% RSLogix 500 project HB_3_Filler.RSS, saved by version 12.00.00.00 %
PROJECT "PLC"    % processor: MicroLogix 1400 %

PROGRAM FILES
  LAD 2   23 rungs
  LAD 9   42 rungs
  LAD 11   37 rungs
  LAD 12   16 rungs
  LAD 14   17 rungs

DATA FILES
  O0 OUTPUT  7 elements
  I1 INPUT  9 elements
  S2 STATUS  66 elements
  B3 BINARY  14 elements
  T4 TIMER  22 elements
  C5 COUNTER  10 elements
  R6 CONTROL  5 elements
  N7 INTEGER  50 elements
  F8 FLOAT  40 elements
  B11   5 elements
  B12   10 elements
  B13   10 elements
  B23   30 elements
  T24   90 elements
  C25   10 elements
  N27   200 elements
  F28   40 elements

LADDER 2
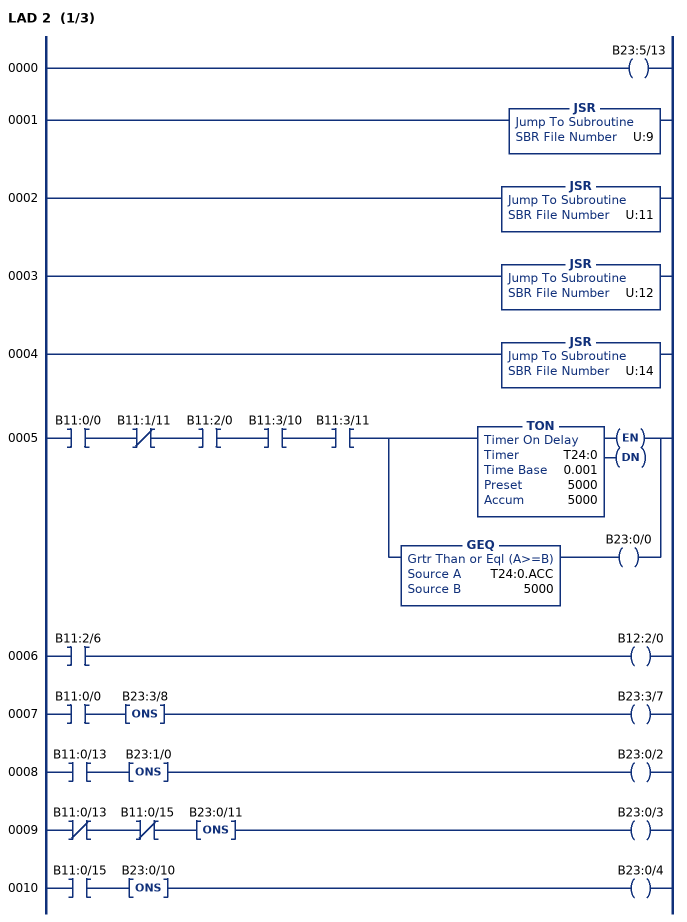
% Rung: 0 %
SOR OTE B23:5/13 EOR
% Rung: 1 %
SOR JSR U:9 EOR
% Rung: 2 %
SOR JSR U:11 EOR
% Rung: 3 %
SOR JSR U:12 EOR
% Rung: 4 %
SOR JSR U:14 EOR
% Rung: 5 %
SOR XIC B11:0/0 XIO B11:1/11 XIC B11:2/0 XIC B11:3/10 XIC B11:3/11 BST TON T24:0 0.001 5000 5000 NXB GEQ T24:0.ACC 5000 OTE B23:0/0 BND EOR
% Rung: 6 %
SOR XIC B11:2/6 OTE B12:2/0 EOR
% Rung: 7 %
SOR XIC B11:0/0 ONS B23:3/8 OTE B23:3/7 EOR
% Rung: 8 %
SOR XIC B11:0/13 ONS B23:1/0 OTE B23:0/2 EOR
% Rung: 9 %
SOR XIO B11:0/13 XIO B11:0/15 ONS B23:0/11 OTE B23:0/3 EOR
% Rung: 10 %
SOR XIC B11:0/15 ONS B23:0/10 OTE B23:0/4 EOR

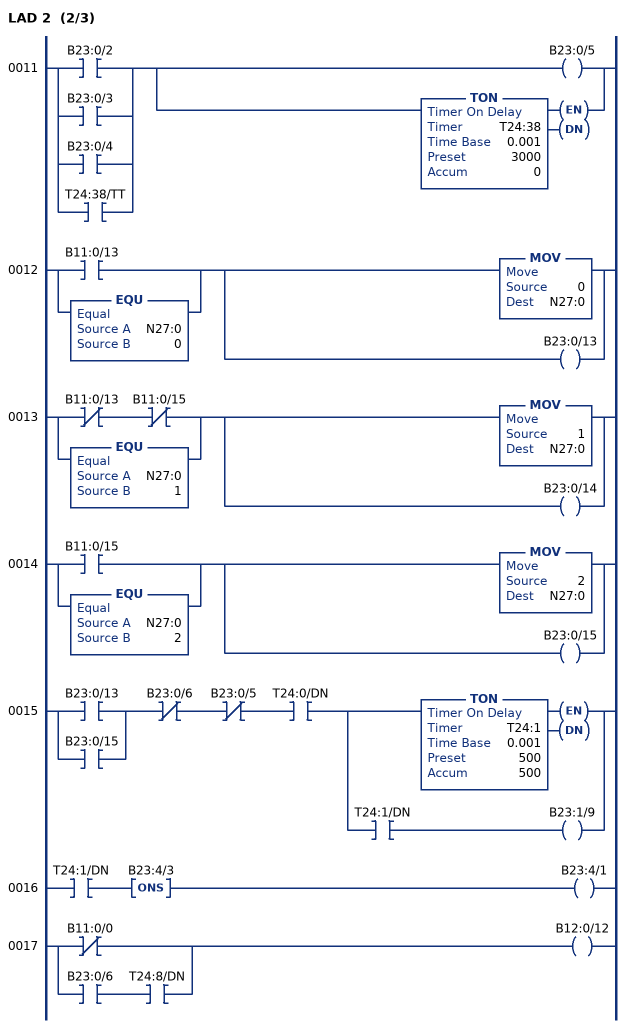
% Rung: 11 %
SOR BST XIC B23:0/2 NXB XIC B23:0/3 NXB XIC B23:0/4 NXB XIC T24:38/TT BND BST OTE B23:0/5 NXB TON T24:38 0.001 3000 0 BND EOR
% Rung: 12 %
SOR BST XIC B11:0/13 NXB EQU N27:0 0 BND BST MOV 0 N27:0 NXB OTE B23:0/13 BND EOR
% Rung: 13 %
SOR BST XIO B11:0/13 XIO B11:0/15 NXB EQU N27:0 1 BND BST MOV 1 N27:0 NXB OTE B23:0/14 BND EOR
% Rung: 14 %
SOR BST XIC B11:0/15 NXB EQU N27:0 2 BND BST MOV 2 N27:0 NXB OTE B23:0/15 BND EOR
% Rung: 15 %
SOR BST XIC B23:0/13 NXB XIC B23:0/15 BND XIO B23:0/6 XIO B23:0/5 XIC T24:0/DN BST TON T24:1 0.001 500 500 NXB XIC T24:1/DN OTE B23:1/9 BND EOR
% Rung: 16 %
SOR XIC T24:1/DN ONS B23:4/3 OTE B23:4/1 EOR
% Rung: 17 %
SOR BST XIO B11:0/0 NXB XIC B23:0/6 XIC T24:8/DN BND OTE B12:0/12 EOR

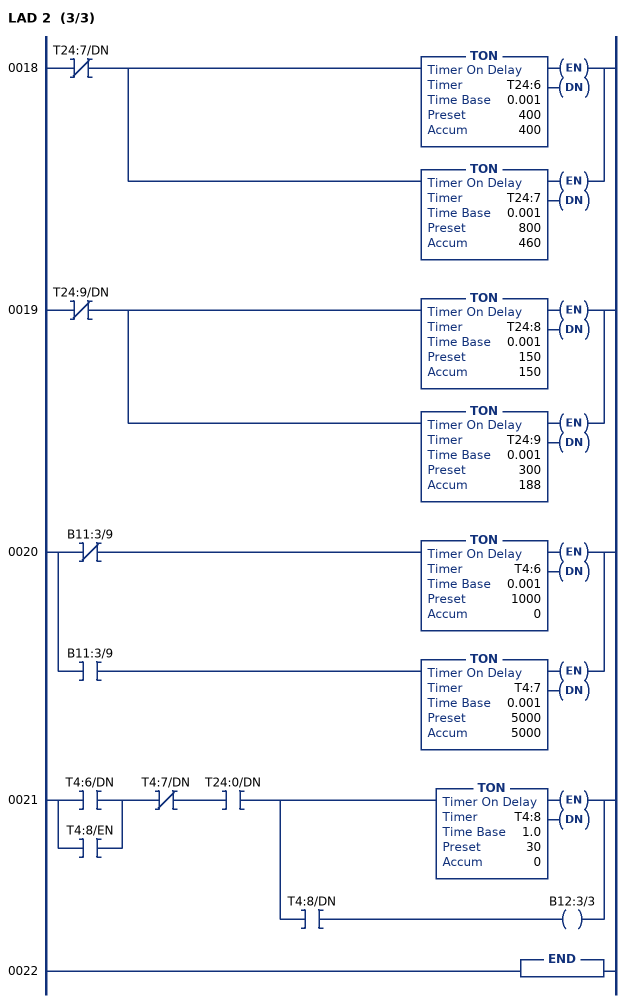
% Rung: 18 %
SOR XIO T24:7/DN BST TON T24:6 0.001 400 400 NXB TON T24:7 0.001 800 460 BND EOR
% Rung: 19 %
SOR XIO T24:9/DN BST TON T24:8 0.001 150 150 NXB TON T24:9 0.001 300 188 BND EOR
% Rung: 20 %
SOR BST XIO B11:3/9 TON T4:6 0.001 1000 0 NXB XIC B11:3/9 TON T4:7 0.001 5000 5000 BND EOR
% Rung: 21 %
SOR BST XIC T4:6/DN NXB XIC T4:8/EN BND XIO T4:7/DN XIC T24:0/DN BST TON T4:8 1.0 30 0 NXB XIC T4:8/DN OTE B12:3/3 BND EOR
% Rung: 22 %
SOR END EOR

LADDER 9
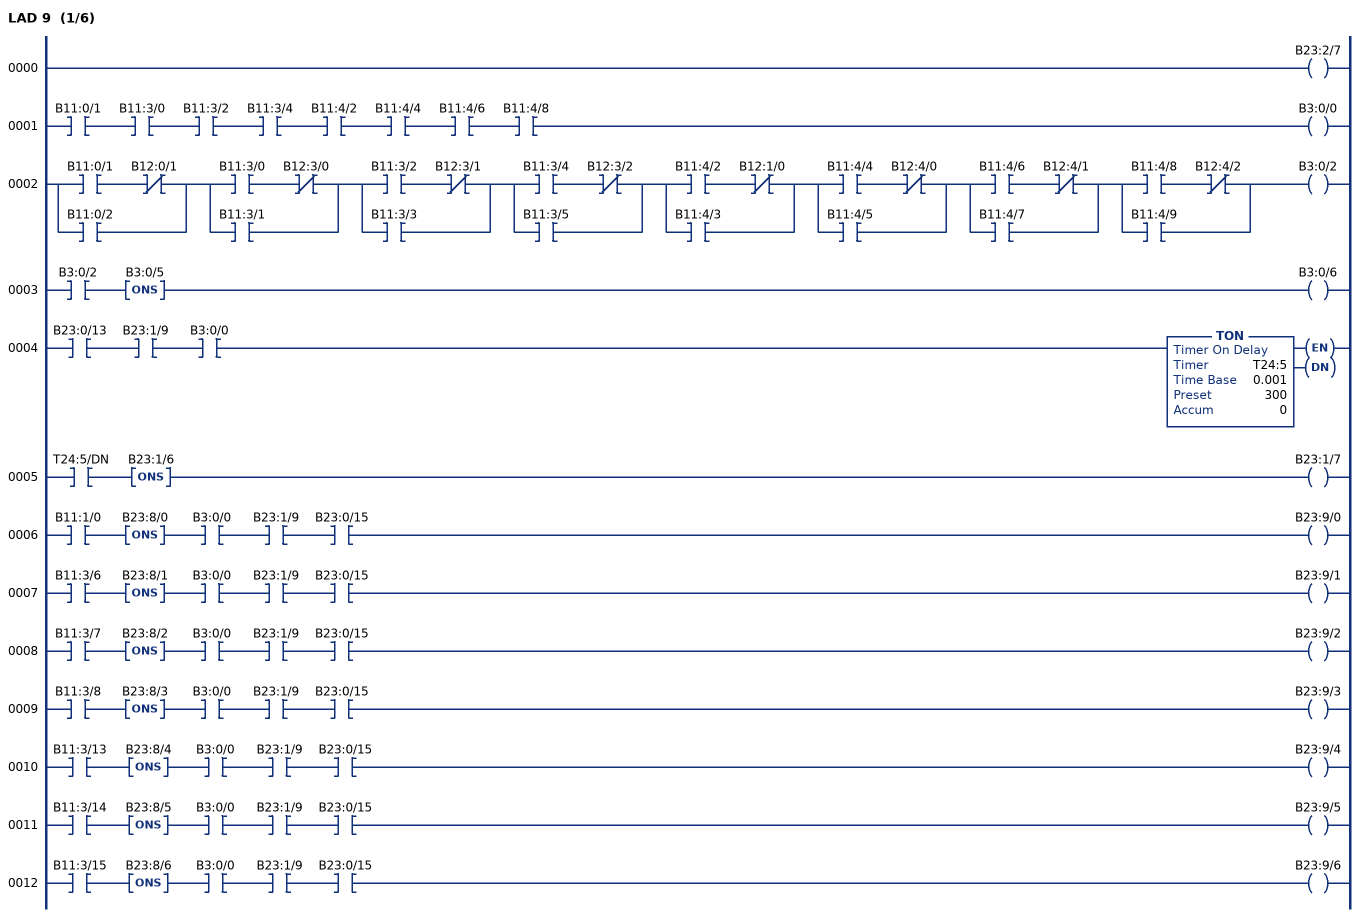
% Rung: 0 %
SOR OTE B23:2/7 EOR
% Rung: 1 %
SOR XIC B11:0/1 XIC B11:3/0 XIC B11:3/2 XIC B11:3/4 XIC B11:4/2 XIC B11:4/4 XIC B11:4/6 XIC B11:4/8 OTE B3:0/0 EOR
% Rung: 2 %
SOR BST XIC B11:0/1 XIO B12:0/1 NXB XIC B11:0/2 BND BST XIC B11:3/0 XIO B12:3/0 NXB XIC B11:3/1 BND BST XIC B11:3/2 XIO B12:3/1 NXB XIC B11:3/3 BND BST XIC B11:3/4 XIO B12:3/2 NXB XIC B11:3/5 BND BST XIC B11:4/2 XIO B12:1/0 NXB XIC B11:4/3 BND BST XIC B11:4/4 XIO B12:4/0 NXB XIC B11:4/5 BND BST XIC B11:4/6 XIO B12:4/1 NXB XIC B11:4/7 BND BST XIC B11:4/8 XIO B12:4/2 NXB XIC B11:4/9 BND OTE B3:0/2 EOR
% Rung: 3 %
SOR XIC B3:0/2 ONS B3:0/5 OTE B3:0/6 EOR
% Rung: 4 %
SOR XIC B23:0/13 XIC B23:1/9 XIC B3:0/0 TON T24:5 0.001 300 0 EOR
% Rung: 5 %
SOR XIC T24:5/DN ONS B23:1/6 OTE B23:1/7 EOR
% Rung: 6 %
SOR XIC B11:1/0 ONS B23:8/0 XIC B3:0/0 XIC B23:1/9 XIC B23:0/15 OTE B23:9/0 EOR
% Rung: 7 %
SOR XIC B11:3/6 ONS B23:8/1 XIC B3:0/0 XIC B23:1/9 XIC B23:0/15 OTE B23:9/1 EOR
% Rung: 8 %
SOR XIC B11:3/7 ONS B23:8/2 XIC B3:0/0 XIC B23:1/9 XIC B23:0/15 OTE B23:9/2 EOR
% Rung: 9 %
SOR XIC B11:3/8 ONS B23:8/3 XIC B3:0/0 XIC B23:1/9 XIC B23:0/15 OTE B23:9/3 EOR
% Rung: 10 %
SOR XIC B11:3/13 ONS B23:8/4 XIC B3:0/0 XIC B23:1/9 XIC B23:0/15 OTE B23:9/4 EOR
% Rung: 11 %
SOR XIC B11:3/14 ONS B23:8/5 XIC B3:0/0 XIC B23:1/9 XIC B23:0/15 OTE B23:9/5 EOR
% Rung: 12 %
SOR XIC B11:3/15 ONS B23:8/6 XIC B3:0/0 XIC B23:1/9 XIC B23:0/15 OTE B23:9/6 EOR

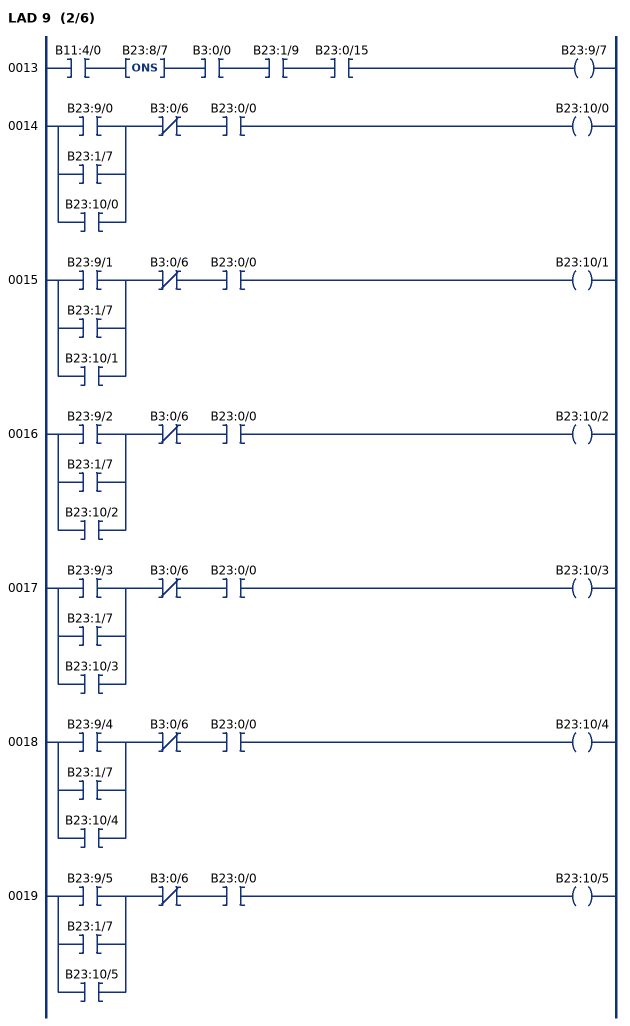
% Rung: 13 %
SOR XIC B11:4/0 ONS B23:8/7 XIC B3:0/0 XIC B23:1/9 XIC B23:0/15 OTE B23:9/7 EOR
% Rung: 14 %
SOR BST XIC B23:9/0 NXB XIC B23:1/7 NXB XIC B23:10/0 BND XIO B3:0/6 XIC B23:0/0 OTE B23:10/0 EOR
% Rung: 15 %
SOR BST XIC B23:9/1 NXB XIC B23:1/7 NXB XIC B23:10/1 BND XIO B3:0/6 XIC B23:0/0 OTE B23:10/1 EOR
% Rung: 16 %
SOR BST XIC B23:9/2 NXB XIC B23:1/7 NXB XIC B23:10/2 BND XIO B3:0/6 XIC B23:0/0 OTE B23:10/2 EOR
% Rung: 17 %
SOR BST XIC B23:9/3 NXB XIC B23:1/7 NXB XIC B23:10/3 BND XIO B3:0/6 XIC B23:0/0 OTE B23:10/3 EOR
% Rung: 18 %
SOR BST XIC B23:9/4 NXB XIC B23:1/7 NXB XIC B23:10/4 BND XIO B3:0/6 XIC B23:0/0 OTE B23:10/4 EOR
% Rung: 19 %
SOR BST XIC B23:9/5 NXB XIC B23:1/7 NXB XIC B23:10/5 BND XIO B3:0/6 XIC B23:0/0 OTE B23:10/5 EOR

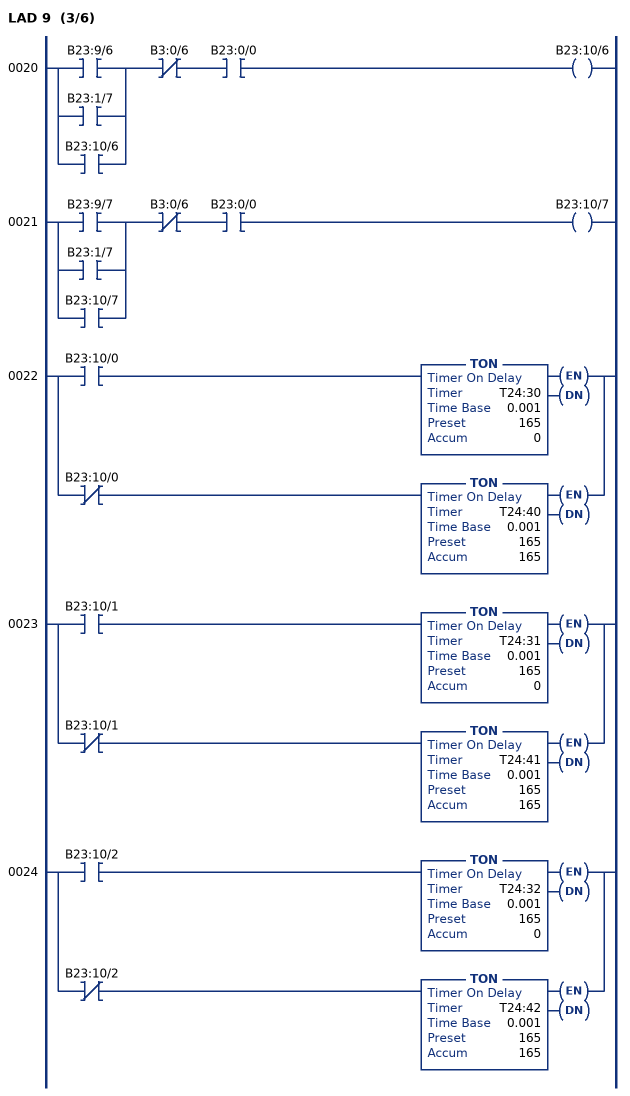
% Rung: 20 %
SOR BST XIC B23:9/6 NXB XIC B23:1/7 NXB XIC B23:10/6 BND XIO B3:0/6 XIC B23:0/0 OTE B23:10/6 EOR
% Rung: 21 %
SOR BST XIC B23:9/7 NXB XIC B23:1/7 NXB XIC B23:10/7 BND XIO B3:0/6 XIC B23:0/0 OTE B23:10/7 EOR
% Rung: 22 %
SOR BST XIC B23:10/0 TON T24:30 0.001 165 0 NXB XIO B23:10/0 TON T24:40 0.001 165 165 BND EOR
% Rung: 23 %
SOR BST XIC B23:10/1 TON T24:31 0.001 165 0 NXB XIO B23:10/1 TON T24:41 0.001 165 165 BND EOR
% Rung: 24 %
SOR BST XIC B23:10/2 TON T24:32 0.001 165 0 NXB XIO B23:10/2 TON T24:42 0.001 165 165 BND EOR

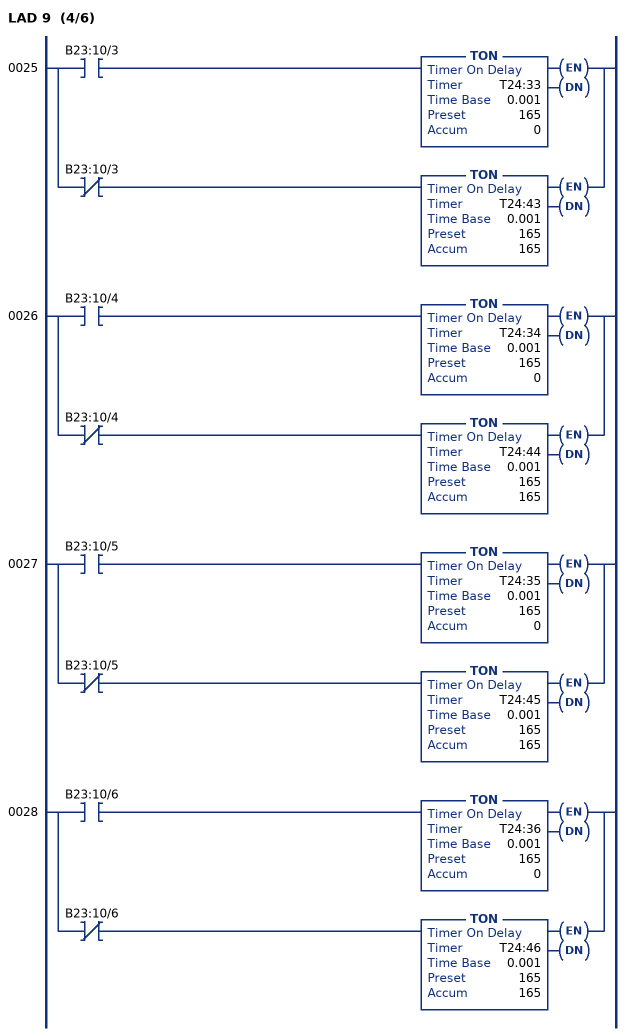
% Rung: 25 %
SOR BST XIC B23:10/3 TON T24:33 0.001 165 0 NXB XIO B23:10/3 TON T24:43 0.001 165 165 BND EOR
% Rung: 26 %
SOR BST XIC B23:10/4 TON T24:34 0.001 165 0 NXB XIO B23:10/4 TON T24:44 0.001 165 165 BND EOR
% Rung: 27 %
SOR BST XIC B23:10/5 TON T24:35 0.001 165 0 NXB XIO B23:10/5 TON T24:45 0.001 165 165 BND EOR
% Rung: 28 %
SOR BST XIC B23:10/6 TON T24:36 0.001 165 0 NXB XIO B23:10/6 TON T24:46 0.001 165 165 BND EOR

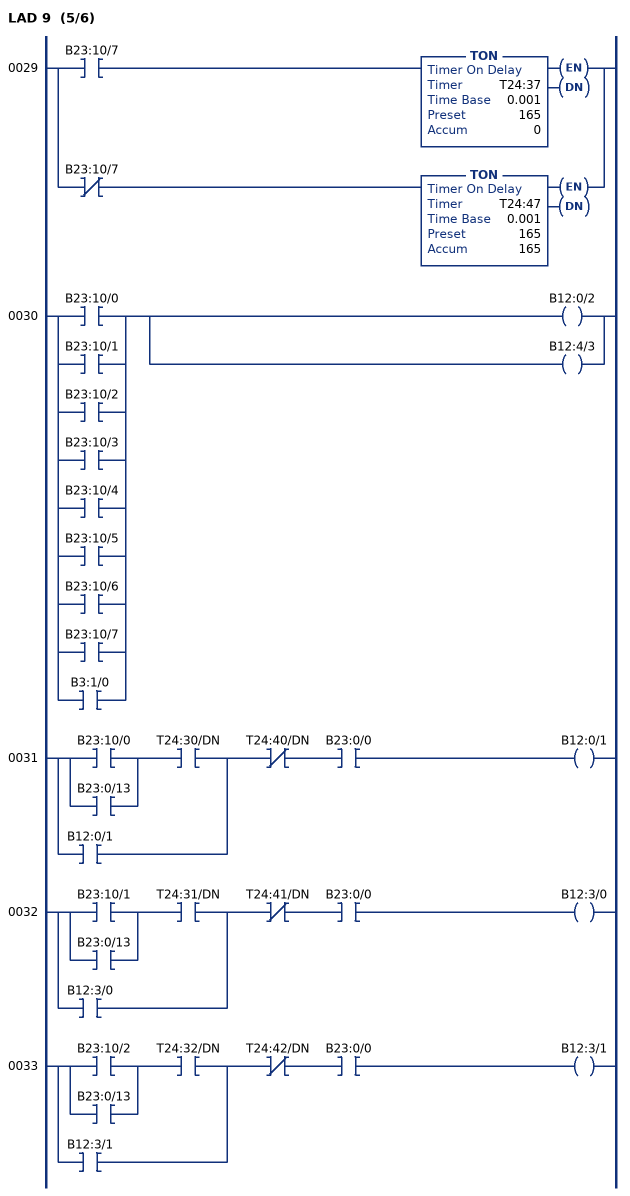
% Rung: 29 %
SOR BST XIC B23:10/7 TON T24:37 0.001 165 0 NXB XIO B23:10/7 TON T24:47 0.001 165 165 BND EOR
% Rung: 30 %
SOR BST XIC B23:10/0 NXB XIC B23:10/1 NXB XIC B23:10/2 NXB XIC B23:10/3 NXB XIC B23:10/4 NXB XIC B23:10/5 NXB XIC B23:10/6 NXB XIC B23:10/7 NXB XIC B3:1/0 BND BST OTE B12:0/2 NXB OTE B12:4/3 BND EOR
% Rung: 31 %
SOR BST BST XIC B23:10/0 NXB XIC B23:0/13 BND XIC T24:30/DN NXB XIC B12:0/1 BND XIO T24:40/DN XIC B23:0/0 OTE B12:0/1 EOR
% Rung: 32 %
SOR BST BST XIC B23:10/1 NXB XIC B23:0/13 BND XIC T24:31/DN NXB XIC B12:3/0 BND XIO T24:41/DN XIC B23:0/0 OTE B12:3/0 EOR
% Rung: 33 %
SOR BST BST XIC B23:10/2 NXB XIC B23:0/13 BND XIC T24:32/DN NXB XIC B12:3/1 BND XIO T24:42/DN XIC B23:0/0 OTE B12:3/1 EOR

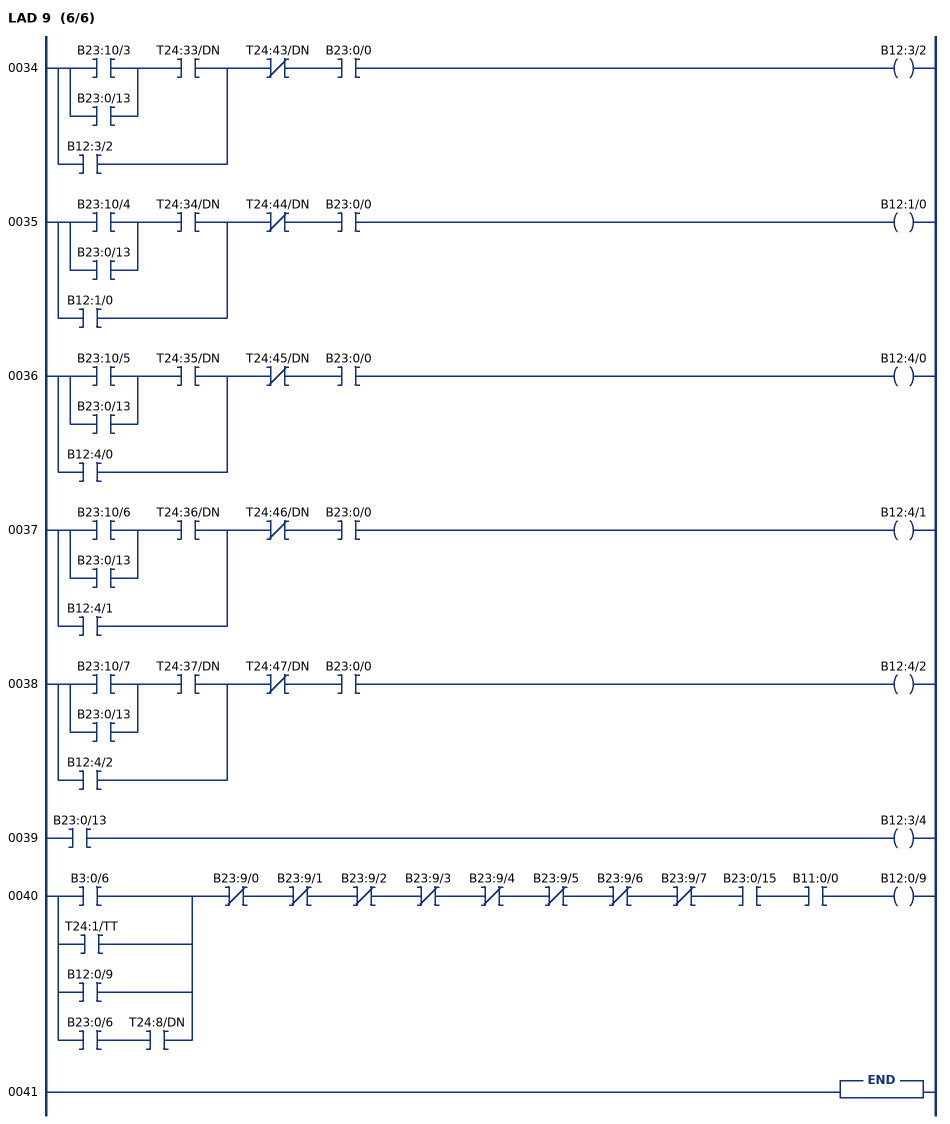
% Rung: 34 %
SOR BST BST XIC B23:10/3 NXB XIC B23:0/13 BND XIC T24:33/DN NXB XIC B12:3/2 BND XIO T24:43/DN XIC B23:0/0 OTE B12:3/2 EOR
% Rung: 35 %
SOR BST BST XIC B23:10/4 NXB XIC B23:0/13 BND XIC T24:34/DN NXB XIC B12:1/0 BND XIO T24:44/DN XIC B23:0/0 OTE B12:1/0 EOR
% Rung: 36 %
SOR BST BST XIC B23:10/5 NXB XIC B23:0/13 BND XIC T24:35/DN NXB XIC B12:4/0 BND XIO T24:45/DN XIC B23:0/0 OTE B12:4/0 EOR
% Rung: 37 %
SOR BST BST XIC B23:10/6 NXB XIC B23:0/13 BND XIC T24:36/DN NXB XIC B12:4/1 BND XIO T24:46/DN XIC B23:0/0 OTE B12:4/1 EOR
% Rung: 38 %
SOR BST BST XIC B23:10/7 NXB XIC B23:0/13 BND XIC T24:37/DN NXB XIC B12:4/2 BND XIO T24:47/DN XIC B23:0/0 OTE B12:4/2 EOR
% Rung: 39 %
SOR XIC B23:0/13 OTE B12:3/4 EOR
% Rung: 40 %
SOR BST XIC B3:0/6 NXB XIC T24:1/TT NXB XIC B12:0/9 NXB XIC B23:0/6 XIC T24:8/DN BND XIO B23:9/0 XIO B23:9/1 XIO B23:9/2 XIO B23:9/3 XIO B23:9/4 XIO B23:9/5 XIO B23:9/6 XIO B23:9/7 XIC B23:0/15 XIC B11:0/0 OTE B12:0/9 EOR
% Rung: 41 %
SOR END EOR

LADDER 11
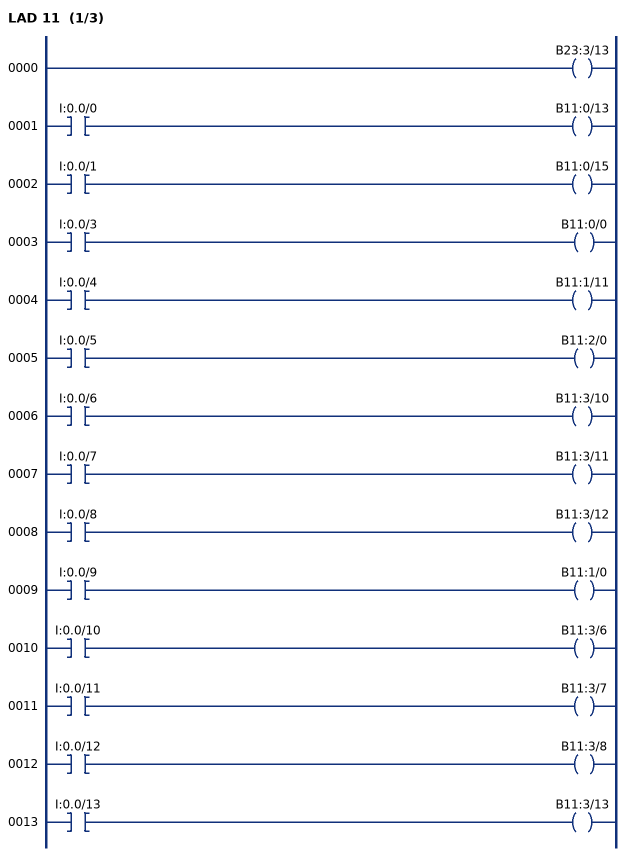
% Rung: 0 %
SOR OTE B23:3/13 EOR
% Rung: 1 %
SOR XIC I:0.0/0 OTE B11:0/13 EOR
% Rung: 2 %
SOR XIC I:0.0/1 OTE B11:0/15 EOR
% Rung: 3 %
SOR XIC I:0.0/3 OTE B11:0/0 EOR
% Rung: 4 %
SOR XIC I:0.0/4 OTE B11:1/11 EOR
% Rung: 5 %
SOR XIC I:0.0/5 OTE B11:2/0 EOR
% Rung: 6 %
SOR XIC I:0.0/6 OTE B11:3/10 EOR
% Rung: 7 %
SOR XIC I:0.0/7 OTE B11:3/11 EOR
% Rung: 8 %
SOR XIC I:0.0/8 OTE B11:3/12 EOR
% Rung: 9 %
SOR XIC I:0.0/9 OTE B11:1/0 EOR
% Rung: 10 %
SOR XIC I:0.0/10 OTE B11:3/6 EOR
% Rung: 11 %
SOR XIC I:0.0/11 OTE B11:3/7 EOR
% Rung: 12 %
SOR XIC I:0.0/12 OTE B11:3/8 EOR
% Rung: 13 %
SOR XIC I:0.0/13 OTE B11:3/13 EOR

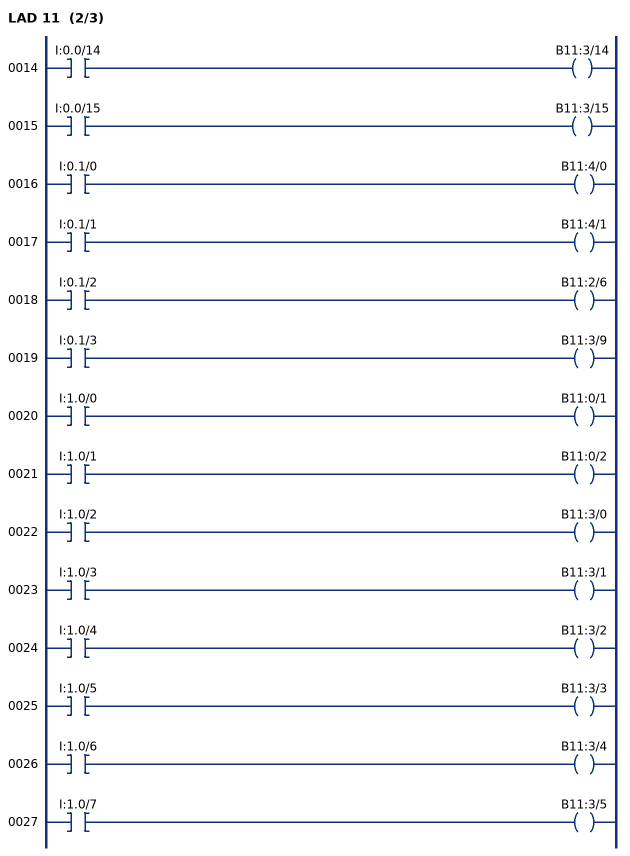
% Rung: 14 %
SOR XIC I:0.0/14 OTE B11:3/14 EOR
% Rung: 15 %
SOR XIC I:0.0/15 OTE B11:3/15 EOR
% Rung: 16 %
SOR XIC I:0.1/0 OTE B11:4/0 EOR
% Rung: 17 %
SOR XIC I:0.1/1 OTE B11:4/1 EOR
% Rung: 18 %
SOR XIC I:0.1/2 OTE B11:2/6 EOR
% Rung: 19 %
SOR XIC I:0.1/3 OTE B11:3/9 EOR
% Rung: 20 %
SOR XIC I:1.0/0 OTE B11:0/1 EOR
% Rung: 21 %
SOR XIC I:1.0/1 OTE B11:0/2 EOR
% Rung: 22 %
SOR XIC I:1.0/2 OTE B11:3/0 EOR
% Rung: 23 %
SOR XIC I:1.0/3 OTE B11:3/1 EOR
% Rung: 24 %
SOR XIC I:1.0/4 OTE B11:3/2 EOR
% Rung: 25 %
SOR XIC I:1.0/5 OTE B11:3/3 EOR
% Rung: 26 %
SOR XIC I:1.0/6 OTE B11:3/4 EOR
% Rung: 27 %
SOR XIC I:1.0/7 OTE B11:3/5 EOR

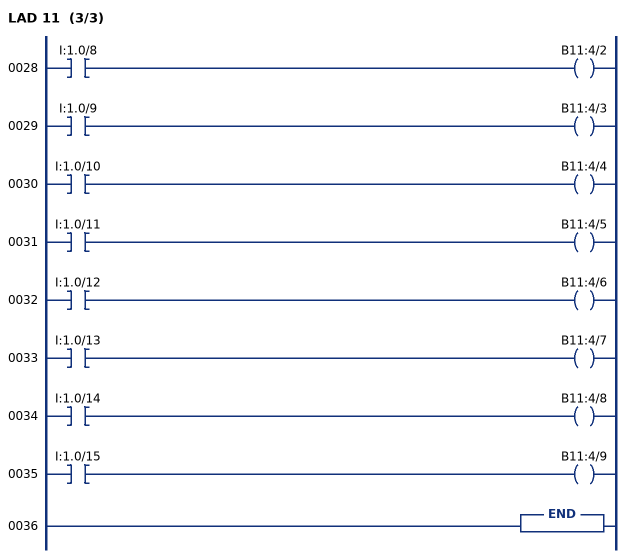
% Rung: 28 %
SOR XIC I:1.0/8 OTE B11:4/2 EOR
% Rung: 29 %
SOR XIC I:1.0/9 OTE B11:4/3 EOR
% Rung: 30 %
SOR XIC I:1.0/10 OTE B11:4/4 EOR
% Rung: 31 %
SOR XIC I:1.0/11 OTE B11:4/5 EOR
% Rung: 32 %
SOR XIC I:1.0/12 OTE B11:4/6 EOR
% Rung: 33 %
SOR XIC I:1.0/13 OTE B11:4/7 EOR
% Rung: 34 %
SOR XIC I:1.0/14 OTE B11:4/8 EOR
% Rung: 35 %
SOR XIC I:1.0/15 OTE B11:4/9 EOR
% Rung: 36 %
SOR END EOR

LADDER 12
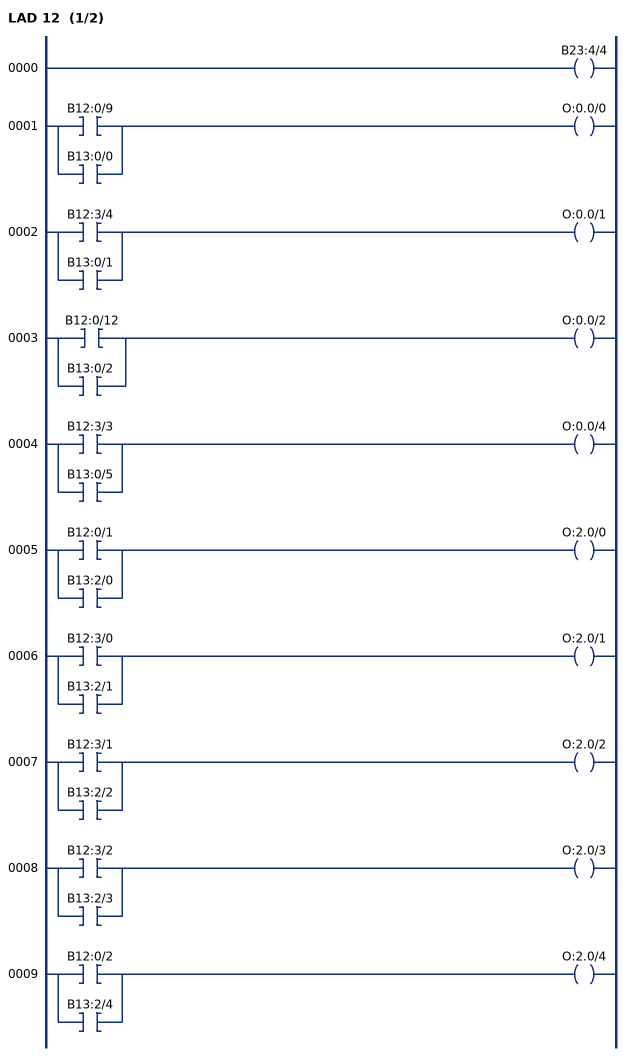
% Rung: 0 %
SOR OTE B23:4/4 EOR
% Rung: 1 %
SOR BST XIC B12:0/9 NXB XIC B13:0/0 BND OTE O:0.0/0 EOR
% Rung: 2 %
SOR BST XIC B12:3/4 NXB XIC B13:0/1 BND OTE O:0.0/1 EOR
% Rung: 3 %
SOR BST XIC B12:0/12 NXB XIC B13:0/2 BND OTE O:0.0/2 EOR
% Rung: 4 %
SOR BST XIC B12:3/3 NXB XIC B13:0/5 BND OTE O:0.0/4 EOR
% Rung: 5 %
SOR BST XIC B12:0/1 NXB XIC B13:2/0 BND OTE O:2.0/0 EOR
% Rung: 6 %
SOR BST XIC B12:3/0 NXB XIC B13:2/1 BND OTE O:2.0/1 EOR
% Rung: 7 %
SOR BST XIC B12:3/1 NXB XIC B13:2/2 BND OTE O:2.0/2 EOR
% Rung: 8 %
SOR BST XIC B12:3/2 NXB XIC B13:2/3 BND OTE O:2.0/3 EOR
% Rung: 9 %
SOR BST XIC B12:0/2 NXB XIC B13:2/4 BND OTE O:2.0/4 EOR

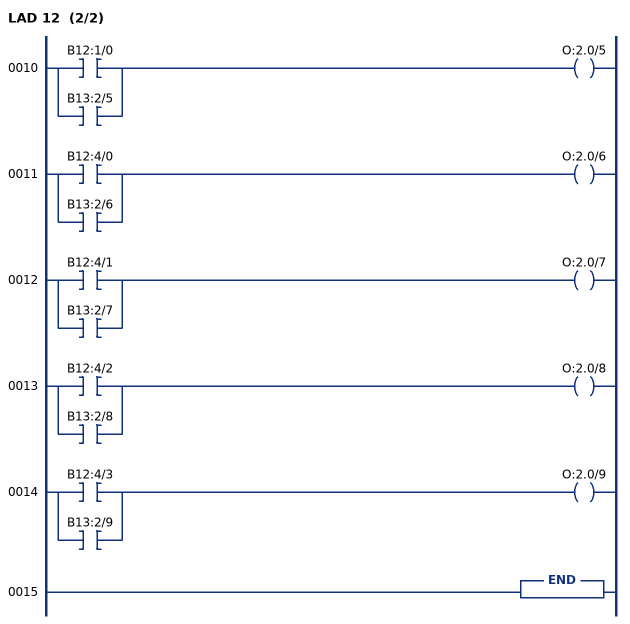
% Rung: 10 %
SOR BST XIC B12:1/0 NXB XIC B13:2/5 BND OTE O:2.0/5 EOR
% Rung: 11 %
SOR BST XIC B12:4/0 NXB XIC B13:2/6 BND OTE O:2.0/6 EOR
% Rung: 12 %
SOR BST XIC B12:4/1 NXB XIC B13:2/7 BND OTE O:2.0/7 EOR
% Rung: 13 %
SOR BST XIC B12:4/2 NXB XIC B13:2/8 BND OTE O:2.0/8 EOR
% Rung: 14 %
SOR BST XIC B12:4/3 NXB XIC B13:2/9 BND OTE O:2.0/9 EOR
% Rung: 15 %
SOR END EOR

LADDER 14
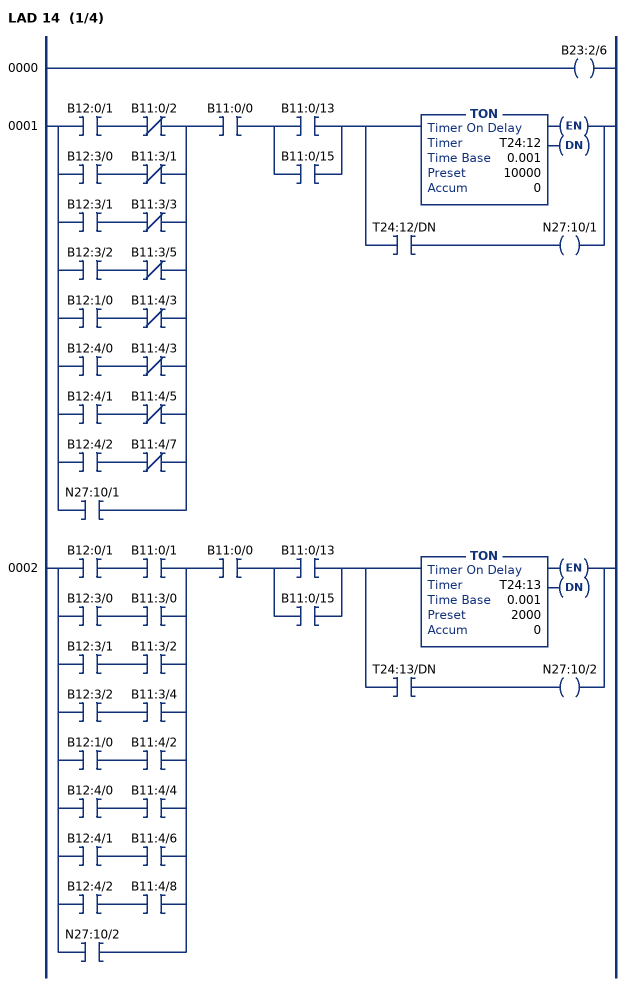
% Rung: 0 %
SOR OTE B23:2/6 EOR
% Rung: 1 %
SOR BST XIC B12:0/1 XIO B11:0/2 NXB XIC B12:3/0 XIO B11:3/1 NXB XIC B12:3/1 XIO B11:3/3 NXB XIC B12:3/2 XIO B11:3/5 NXB XIC B12:1/0 XIO B11:4/3 NXB XIC B12:4/0 XIO B11:4/3 NXB XIC B12:4/1 XIO B11:4/5 NXB XIC B12:4/2 XIO B11:4/7 NXB XIC N27:10/1 BND XIC B11:0/0 BST XIC B11:0/13 NXB XIC B11:0/15 BND BST TON T24:12 0.001 10000 0 NXB XIC T24:12/DN OTE N27:10/1 BND EOR
% Rung: 2 %
SOR BST XIC B12:0/1 XIC B11:0/1 NXB XIC B12:3/0 XIC B11:3/0 NXB XIC B12:3/1 XIC B11:3/2 NXB XIC B12:3/2 XIC B11:3/4 NXB XIC B12:1/0 XIC B11:4/2 NXB XIC B12:4/0 XIC B11:4/4 NXB XIC B12:4/1 XIC B11:4/6 NXB XIC B12:4/2 XIC B11:4/8 NXB XIC N27:10/2 BND XIC B11:0/0 BST XIC B11:0/13 NXB XIC B11:0/15 BND BST TON T24:13 0.001 2000 0 NXB XIC T24:13/DN OTE N27:10/2 BND EOR

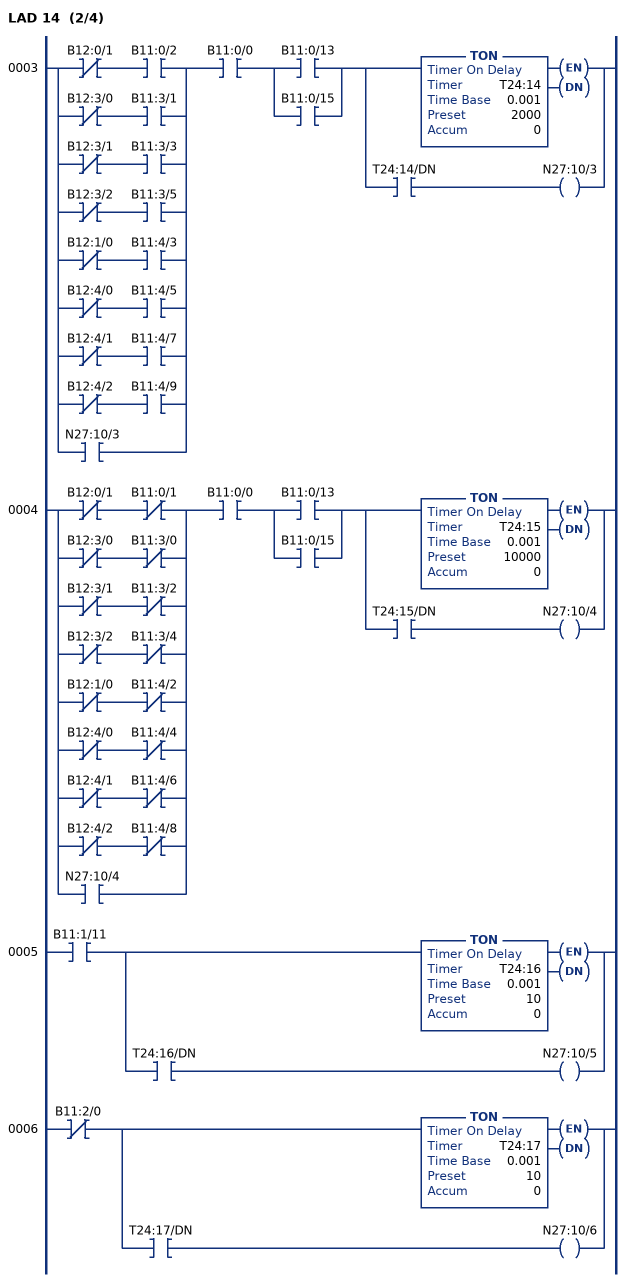
% Rung: 3 %
SOR BST XIO B12:0/1 XIC B11:0/2 NXB XIO B12:3/0 XIC B11:3/1 NXB XIO B12:3/1 XIC B11:3/3 NXB XIO B12:3/2 XIC B11:3/5 NXB XIO B12:1/0 XIC B11:4/3 NXB XIO B12:4/0 XIC B11:4/5 NXB XIO B12:4/1 XIC B11:4/7 NXB XIO B12:4/2 XIC B11:4/9 NXB XIC N27:10/3 BND XIC B11:0/0 BST XIC B11:0/13 NXB XIC B11:0/15 BND BST TON T24:14 0.001 2000 0 NXB XIC T24:14/DN OTE N27:10/3 BND EOR
% Rung: 4 %
SOR BST XIO B12:0/1 XIO B11:0/1 NXB XIO B12:3/0 XIO B11:3/0 NXB XIO B12:3/1 XIO B11:3/2 NXB XIO B12:3/2 XIO B11:3/4 NXB XIO B12:1/0 XIO B11:4/2 NXB XIO B12:4/0 XIO B11:4/4 NXB XIO B12:4/1 XIO B11:4/6 NXB XIO B12:4/2 XIO B11:4/8 NXB XIC N27:10/4 BND XIC B11:0/0 BST XIC B11:0/13 NXB XIC B11:0/15 BND BST TON T24:15 0.001 10000 0 NXB XIC T24:15/DN OTE N27:10/4 BND EOR
% Rung: 5 %
SOR XIC B11:1/11 BST TON T24:16 0.001 10 0 NXB XIC T24:16/DN OTE N27:10/5 BND EOR
% Rung: 6 %
SOR XIO B11:2/0 BST TON T24:17 0.001 10 0 NXB XIC T24:17/DN OTE N27:10/6 BND EOR

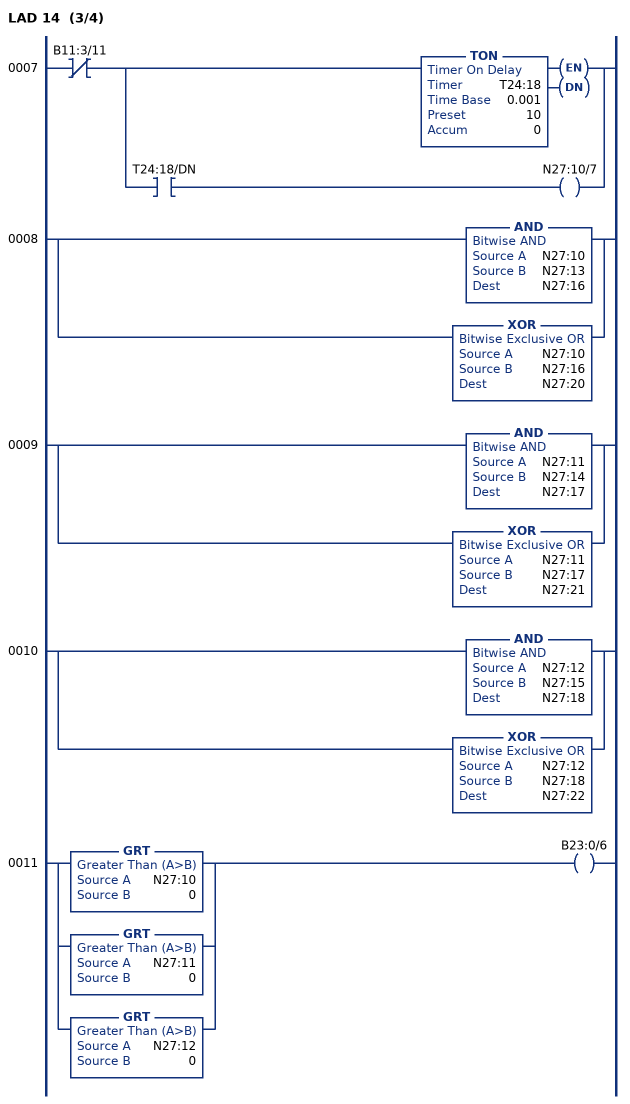
% Rung: 7 %
SOR XIO B11:3/11 BST TON T24:18 0.001 10 0 NXB XIC T24:18/DN OTE N27:10/7 BND EOR
% Rung: 8 %
SOR BST AND N27:10 N27:13 N27:16 NXB XOR N27:10 N27:16 N27:20 BND EOR
% Rung: 9 %
SOR BST AND N27:11 N27:14 N27:17 NXB XOR N27:11 N27:17 N27:21 BND EOR
% Rung: 10 %
SOR BST AND N27:12 N27:15 N27:18 NXB XOR N27:12 N27:18 N27:22 BND EOR
% Rung: 11 %
SOR BST GRT N27:10 0 NXB GRT N27:11 0 NXB GRT N27:12 0 BND OTE B23:0/6 EOR

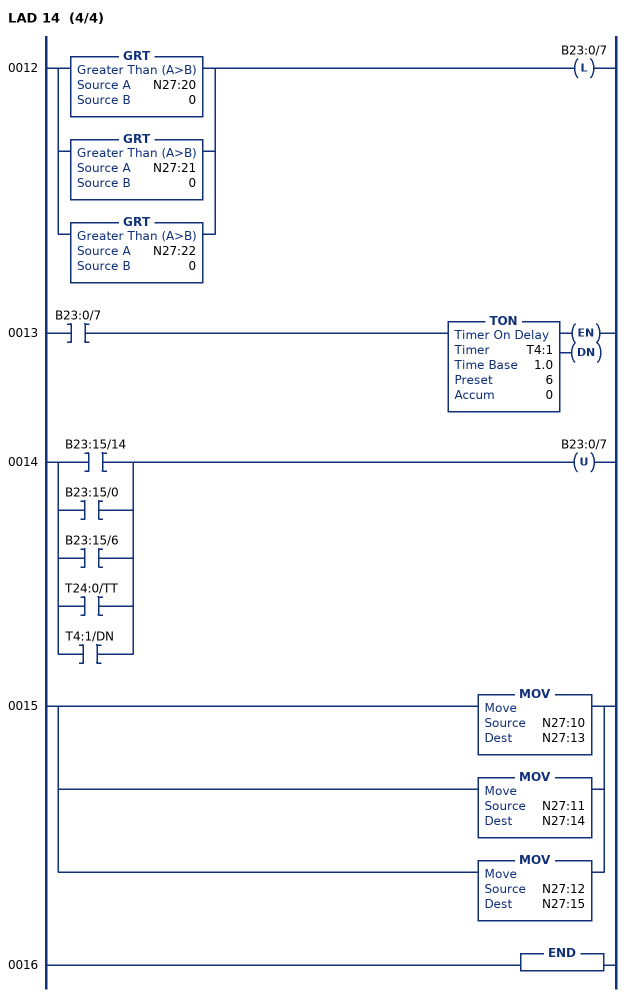
% Rung: 12 %
SOR BST GRT N27:20 0 NXB GRT N27:21 0 NXB GRT N27:22 0 BND OTL B23:0/7 EOR
% Rung: 13 %
SOR XIC B23:0/7 TON T4:1 1.0 6 0 EOR
% Rung: 14 %
SOR BST XIC B23:15/14 NXB XIC B23:15/0 NXB XIC B23:15/6 NXB XIC T24:0/TT NXB XIC T4:1/DN BND OTU B23:0/7 EOR
% Rung: 15 %
SOR BST MOV N27:10 N27:13 NXB MOV N27:11 N27:14 NXB MOV N27:12 N27:15 BND EOR
% Rung: 16 %
SOR END EOR

DATA TABLE (non-zero values as saved)
DATA B3
% B3:0 % 0X00BF 0X0004 0X0040 0X0000 0X0000 0X0000 0X0000 0X0000 0X0000 0X0000
DATA T4
% .PRE .ACC %
% T4:0 % 200 0
% T4:1 % 6 0
% T4:2 % 400 0
% T4:3 % 200 0
% T4:4 % 200 0
% T4:5 % 200 200
% T4:6 % 1000 0
% T4:7 % 5000 5000
% T4:8 % 30 0
% T4:9 % 1000 0
% T4:10 % 1000 0
% T4:11 % 300 0
% T4:12 % 300 0
% T4:13 % 300 0
% T4:14 % 300 0
% T4:21 % 10000 0
DATA C5
% .PRE .ACC %
% C5:0 % 4 1
% C5:1 % 10 8
% C5:3 % 99 0
DATA R6
% .LEN .POS %
% R6:0 % 20 0
% R6:1 % 48 0
% R6:2 % 10 9
% R6:3 % 10 9
DATA N7
% N7:0 % 1 131 132 132 133 129 133 131 136 133
% N7:10 % 0 8 0 0 0 0 0 0 0 0
% N7:20 % 0 83 82 81 83 81 82 81 82 82
DATA F8
% F8:0 % 693 550 8 0 0
DATA B11
% B11:0 % 0XDBFB 0X1040 0X0099 0X0E15 0X0154
DATA B12
% B12:0 % 0X46C0 0X0002 0X0000 0X1000 0X0000 0X0000 0X0000 0X0000 0X0000 0X0000
DATA B23
% B23:0 % 0X8401 0X6204 0XBBE0 0X3311 0X21FC 0X2000 0X0000 0X0000 0X0000 0X0000
% B23:10 % 0X0000 0X0000 0X0000 0X0000 0X0000 0X0008 0X0000 0X0000 0X0000 0X0000
DATA T24
% .PRE .ACC %
% T24:0 % 5000 5000
% T24:1 % 500 500
% T24:2 % 2000 0
% T24:3 % 200 0
% T24:4 % 200 200
% T24:5 % 300 0
% T24:6 % 400 400
% T24:7 % 800 460
% T24:8 % 150 150
% T24:9 % 300 188
% T24:10 % 60 52
% T24:11 % 1000 0
% T24:12 % 10000 0
% T24:13 % 2000 0
% T24:14 % 2000 0
% T24:15 % 10000 0
% T24:16 % 10 0
% T24:17 % 10 0
% T24:18 % 10 0
% T24:19 % 2000 0
% T24:20 % 3000 0
% T24:21 % 1000 0
% T24:22 % 1000 0
% T24:23 % 1000 0
% T24:24 % 1000 0
% T24:25 % 1000 0
% T24:26 % 1000 0
% T24:27 % 1000 0
% T24:28 % 1000 0
% T24:29 % 1000 0
% T24:30 % 165 0
% T24:31 % 165 0
% T24:32 % 165 0
% T24:33 % 165 0
% T24:34 % 165 0
% T24:35 % 165 0
% T24:36 % 165 0
% T24:37 % 165 0
% T24:38 % 3000 0
% T24:39 % 500 500
% T24:40 % 165 165
% T24:41 % 165 165
% T24:42 % 165 165
% T24:43 % 165 165
% T24:44 % 165 165
% T24:45 % 165 165
% T24:46 % 165 165
% T24:47 % 165 165
% T24:48 % 10 0
% T24:49 % 3000 0
% T24:50 % 3000 0
% T24:51 % 3000 0
% T24:52 % 100 0
% T24:53 % 200 0
% T24:54 % 10000 0
% T24:55 % 5000 0
% T24:56 % 500 0
% T24:57 % 500 500
% T24:58 % 12000 12000
% T24:60 % 300 0
% T24:65 % 140 0
% T24:69 % 140 0
% T24:72 % 2 0
% T24:82 % 400 400
DATA C25
% .PRE .ACC %
% C25:0 % 1000 0
% C25:1 % 1 0
% C25:2 % 15 0
% C25:3 % 12 1
% C25:5 % 10 0
DATA N27
% N27:0 % 2 2 20 2 1 7 150 150 1 0
% N27:40 % 0 111 222 333 444 555 11112 0 10101 32767
% N27:100 % 0 1 2 3 88 99 99 99 99 99
% N27:110 % 0 99 99 99 99 99 99 99 99 99
% N27:120 % 0 99 99 99 99 99 99 99 99 99
% N27:130 % 0 99 99 99 99 99 99 99 99 99
% N27:140 % 0 99 99 99 99 99 99 99 99 99
% N27:150 % 0 99 99 99 99 99 99 99 99 99
% N27:160 % 0 99 99 99 99 99 99 99 99 99
% N27:170 % 90 99 99 99 99 99 99 99 99 99
DATA F28
% F28:0 % 1 1 1 1 4096
% F28:5 % 25000 0 0 0 0
% F28:10 % 99 250 399 98 0
% F28:20 % 3566 0 0 0 0
